FUNCTION calcPreciseDiff : PtPreciseDiff
VAR_INPUT
	D1 : PtDateTime;
	D2 : PtDateTime;
END_VAR
VAR
	HourDiff : DINT;
	
END_VAR

IF isDateTimeEqual(D1, D2) THEN
	calcPreciseDiff.Set(0,0,0,0,0,0,0,0);
	RETURN;
END_IF
calcPreciseDiff.total_days := ABS(calcDayNumber(D1.Year, d1.Month, d1.Day) - calcDayNumber(D2.Year, d2.Month, d2.Day));

END_FUNCTION

(* stored: Version 1.1.0.1, ProductVersion 3.1.4024.12
   POU calcPreciseDiff: Id {7e667af7-763f-4ef5-baf0-511b98e984ce}, SpecialFunc None *)
